Fanuc KAREL source: port_MRK.kl

PROGRAM TP
%NOLOCKGROUP
VAR
 x: BOOLEAN
BEGIN
 x = MRK[3]
END TP
